{attribute 'qualified_only'}
VAR_GLOBAL
    mb_Input_Coils 				: ARRAY [0..255] OF BOOL;
    mb_Output_Coils 			: ARRAY [0..255] OF BOOL;
    mb_Output_Registers 		: ARRAY [0..255] OF WORD;
    mb_Input_Registers 			: ARRAY [0..255] OF WORD;
END_VAR

(* stored: Version 1.1.0.1
   GVL GVL: Id {d0381540-e73e-49cb-9733-1a4771c062d6} *)
